// TIA Portal project "SUW_NOWE" (V18)

(* hardware
DEVICE "S7-1200 station_1"  S7-1200 Station
   slot 0: "Rack_0"  S7-1200 Rack  Rack  V1.0
   slot 1: "SUW_NOWE_CPU"  CPU 1215C DC/DC/DC  6ES7 215-1AG40-0XB0  V4.4
   slot 2: "DI 8/DQ 8x24VDC_1"  6ES7 223-1BH32-0XB0  V2.0
   slot 3: "AI 8x13BIT_1"  6ES7 231-4HF32-0XB0  V2.1
*)

// ===== PLC "SUW_NOWE_CPU"  CPU 1215C DC/DC/DC =====

VAR_GLOBAL   // PLC tag table "Default tag table"
   "System_Byte" AT %MB1 : Byte;
   "FirstScan" AT %M1.0 : Bool;
   "DiagStatusUpdate" AT %M1.1 : Bool;
   "AlwaysTRUE" AT %M1.2 : Bool;
   "AlwaysFALSE" AT %M1.3 : Bool;
   "Clock_Byte" AT %MB0 : Byte;
   "Clock_10Hz" AT %M0.0 : Bool;
   "Clock_5Hz" AT %M0.1 : Bool;
   "Clock_2.5Hz" AT %M0.2 : Bool;
   "Clock_2Hz" AT %M0.3 : Bool;
   "Clock_1.25Hz" AT %M0.4 : Bool;
   "Clock_1Hz" AT %M0.5 : Bool;
   "Clock_0.625Hz" AT %M0.6 : Bool;
   "Clock_0.5Hz" AT %M0.7 : Bool;
   "ilosc_pomp" AT %MW2 : Int;
   "moc_pomp" AT %MD4 : Real;
   "pomocnicza" AT %M8.0 : Bool;
   "bPumpsEnable" AT %M8.1 : Bool;
   "iNumPumps" AT %MW10 : Int;
   "rPumpSpeed" AT %MD12 : Real;
   "temp" AT %M8.2 : Bool;
   "temp2" AT %M8.3 : Bool;
   "bReadComplet1A" AT %M8.4 : Bool;
   "bReq1A" AT %M8.5 : Bool;
   "bReq2A" AT %M8.6 : Bool;
   "bReadComplet2A" AT %M8.7 : Bool;
   "bReq3A" AT %M9.0 : Bool;
   "bReadComplet3A" AT %M9.1 : Bool;
   "bReq2B" AT %M9.2 : Bool;
   "bReadComplet2B" AT %M9.3 : Bool;
   "bReq3" AT %M9.4 : Bool;
   "bReadComplet3" AT %M9.5 : Bool;
   "bReq5" AT %M9.6 : Bool;
   "bReadComplet5" AT %M9.7 : Bool;
END_VAR

VAR_GLOBAL   // PLC tag table "I/O"
   "bPmp1A_AutoSwitch" AT %I0.0 : Bool;   // Przełącznik AUTO pompy 1A
   "bPmp2A_AutoSwitch" AT %I0.1 : Bool;   // Przełącznik AUTO pompy 2A
   "bPmp2B_AutoSwitch" AT %I0.2 : Bool;   // Przełącznik AUTO pompy 2B
   "bPmp3_AutoSwitch" AT %I0.3 : Bool;   // Przełącznik AUTO pompy 3
   "bPmp3A_AutoSwitch" AT %I0.4 : Bool;   // Przełącznik AUTO pompy 3A
   "bPmp5_AutoSwitch" AT %I0.5 : Bool;   // Przełącznik AUTO pompy 5
   "bPmp1A_ManualSwitch" AT %I1.0 : Bool;   // Przełącznik ręczny pompy 1A
   "bPmp2A_ManualSwitch" AT %I1.1 : Bool;   // Przełącznik ręczny pompy 2A
   "bPmp2B_ManualSwitch" AT %I1.2 : Bool;   // Przełącznik ręczny pompy 2B
   "bPmp3_ManualSwitch" AT %I1.3 : Bool;   // Przełącznik ręczny pompy 3
   "bPmp3A_ManualSwitch" AT %I1.4 : Bool;   // Przełącznik ręczny pompy 3A
   "bPmp5_ManualSwitch" AT %I1.5 : Bool;   // Przełącznik ręczny pompy 5
   "bPmp1A_RunSignal" AT %Q0.0 : Bool;   // Sygnalizacja pracy pompy 1A
   "bPmp2A_RunSignal" AT %Q0.1 : Bool;   // Sygnalizacja pracy pompy 2A
   "bPmp2B_RunSignal" AT %Q0.2 : Bool;   // Sygnalizacja pracy pompy 2B
   "bPmp3_RunSignal" AT %Q0.3 : Bool;   // Sygnalizacja pracy pompy 3
   "bPmp3A_RunSignal" AT %Q0.4 : Bool;   // Sygnalizacja pracy pompy 3A
   "bPmp5_RunSignal" AT %Q0.5 : Bool;   // Sygnalizacja pracy pompy 5
   "bPmp1A_FaultSignal" AT %Q0.6 : Bool;   // Sygnalizacja awarii pompy 1A
   "bPmp2A_FaultSignal" AT %Q0.7 : Bool;   // Sygnalizacja awarii pompy 2A
   "bPmp2B_FaultSignal" AT %Q1.0 : Bool;   // Sygnalizacja awarii pompy 2B
   "bPmp3_FaultSignal" AT %Q1.1 : Bool;   // Sygnalizacja awarii pompy 3
   "bPmp3A_FaultSignal" AT %Q8.0 : Bool;   // Sygnalizacja awarii pompy 3A
   "bPmp5_FaultSignal" AT %Q8.1 : Bool;   // Sygnalizacja awarii pompy 5
END_VAR

DATA_BLOCK "KomunikacjaFalownik1A_DB"   // DB1
{ S7_Optimized_Access := 'TRUE' }
VERSION : 0.1
// stored: InstanceOfName KomunikacjaFalownik
"KomunikacjaFalownik"
BEGIN
END_DATA_BLOCK

DATA_BLOCK "ObslugaGotowosciPompy_1A_DB"   // DB2
{ S7_Optimized_Access := 'TRUE' }
VERSION : 0.1
// stored: InstanceOfName ObslugaGotowosciPompy
"ObslugaGotowosciPompy"
BEGIN
END_DATA_BLOCK

DATA_BLOCK "ObslugaGotowosciPompy_2A_DB"   // DB3
{ S7_Optimized_Access := 'TRUE' }
VERSION : 0.1
// stored: InstanceOfName ObslugaGotowosciPompy
"ObslugaGotowosciPompy"
BEGIN
END_DATA_BLOCK

DATA_BLOCK "ObslugaGotowosciPompy_2B_DB"   // DB4
{ S7_Optimized_Access := 'TRUE' }
VERSION : 0.1
// stored: InstanceOfName ObslugaGotowosciPompy
"ObslugaGotowosciPompy"
BEGIN
END_DATA_BLOCK

DATA_BLOCK "ObslugaGotowosciPompy_3_DB"   // DB5
{ S7_Optimized_Access := 'TRUE' }
VERSION : 0.1
// stored: InstanceOfName ObslugaGotowosciPompy
"ObslugaGotowosciPompy"
BEGIN
END_DATA_BLOCK

DATA_BLOCK "ObslugaGotowosciPompy_3A_DB"   // DB6
{ S7_Optimized_Access := 'TRUE' }
VERSION : 0.1
// stored: InstanceOfName ObslugaGotowosciPompy
"ObslugaGotowosciPompy"
BEGIN
END_DATA_BLOCK

DATA_BLOCK "ObslugaWyboruPomp_DB"   // DB7
{ S7_Optimized_Access := 'TRUE' }
VERSION : 0.1
// stored: InstanceOfName ObslugaWyboruPomp
"ObslugaWyboruPomp"
BEGIN
END_DATA_BLOCK

DATA_BLOCK "AutoReady"   // DB10
{ S7_Optimized_Access := 'TRUE' }
VERSION : 0.1
   VAR
      aReadyArray : Array[1..6] of Bool;
      aPumpToActive : Array[1..6] of Bool;
      iLastRotationTime : DTL;
      aTimePump : Array[1..6] of DInt;
   END_VAR
BEGIN
END_DATA_BLOCK

DATA_BLOCK "MODBUS_SERVER"   // DB11
{ S7_Optimized_Access := 'TRUE' }
VERSION : 0.1
   VAR
      tcp : TCON_IP_v4;
   END_VAR
BEGIN
   tcp.InterfaceId := 64;
   tcp.ID := 16#1;
   tcp.RemotePort := 0;
   tcp.LocalPort := 502;
   tcp.RemoteAddress.ADDR[1] := 192;
   tcp.RemoteAddress.ADDR[2] := 168;
   tcp.RemoteAddress.ADDR[3] := 99;
   tcp.RemoteAddress.ADDR[4] := 200;
   tcp.ActiveEstablished := false;
END_DATA_BLOCK

DATA_BLOCK "KomunikacjaFalownik2A_DB"   // DB13
{ S7_Optimized_Access := 'TRUE' }
VERSION : 0.1
// stored: InstanceOfName KomunikacjaFalownik
"KomunikacjaFalownik"
BEGIN
END_DATA_BLOCK

DATA_BLOCK "KomunikacjaFalownik3A_DB"   // DB14
{ S7_Optimized_Access := 'TRUE' }
VERSION : 0.1
// stored: InstanceOfName KomunikacjaFalownik
"KomunikacjaFalownik"
BEGIN
END_DATA_BLOCK

DATA_BLOCK "KomunikacjaFalownik2B_DB"   // DB17
{ S7_Optimized_Access := 'TRUE' }
VERSION : 0.1
// stored: InstanceOfName KomunikacjaFalownik
"KomunikacjaFalownik"
BEGIN
END_DATA_BLOCK

DATA_BLOCK "KomunikacjaFalownik3_DB"   // DB18
{ S7_Optimized_Access := 'TRUE' }
VERSION : 0.1
// stored: InstanceOfName KomunikacjaFalownik
"KomunikacjaFalownik"
BEGIN
END_DATA_BLOCK

DATA_BLOCK "KomunikacjaFalownik5_DB"   // DB20
{ S7_Optimized_Access := 'TRUE' }
VERSION : 0.1
// stored: InstanceOfName KomunikacjaFalownik
"KomunikacjaFalownik"
BEGIN
END_DATA_BLOCK

DATA_BLOCK "IPBlock"   // DB30
{ S7_Optimized_Access := 'TRUE' }
VERSION : 0.1
   VAR RETAIN
      IP1A : Array[1..4] of Byte;
      IP2A : Array[1..4] of Byte;
      IP2B : Array[1..4] of Byte;
      IP3 : Array[1..4] of Byte;
      IP3A : Array[1..4] of Byte;
      IP5 : Array[1..4] of Byte;
      IPBudynek : Array[1..4] of Byte;
      IPRozdzielnia : Array[1..4] of Byte;
      IPKosiby : Array[1..4] of Byte;
   END_VAR
BEGIN
   IP1A[1] := 192;
   IP1A[2] := 168;
   IP1A[3] := 99;
   IP1A[4] := 111;
   IP2A[1] := 192;
   IP2A[2] := 168;
   IP2A[3] := 99;
   IP2A[4] := 112;
END_DATA_BLOCK

DATA_BLOCK "Studnia1A"   // DB31
{ S7_Optimized_Access := 'FALSE' }
VERSION : 0.1
   VAR
      CONTROL_WORD : Int;   // Słowo sterujące dla falownika
      SETPOINT_R : Real;   // Setpoint w procentach
      SETPOINT : Int;   // Setpoint w wartości dla falownika 0-8333 dla predkości 0-3000 rpm
      STATUS_WORD : Int;   // Słowo statusowe falownika
      ACTUAL_VALUE : Int;   // Aktualna wartość z falownika
      POWER : Int;   // Moc pompy w kW [*0,01]
      MOTOR_CURRENT : Int;   // Prąd pompy w A [*0,01]
      HEATSNK_TEMP : Int;   // Temperatura radiatora w C
      INVERTER_TERM : Int;   // Status termiczny invertera
      ANALOGIN_53 : Int;   // Pętla analogowa 4-20mA (poziom)
      ALARM_WORD : Word;   // Słowo alarmowe
      ALARM_WORD_1 : Word;   // Słowo alarmowe
      ALARM_WORD_2 : Word;   // Słowo alarmowe
      WARNING_WORD : Word;   // Słowo ostrzeżenia
      WARNING_WORD_1 : Word;   // Słowo ostrzeżenia
      WARNING_WORD_2 : Word;   // Słowo ostrzeżenia
      STATUS : Word;   // Status pompy wg. rozpiski
      DONE : Bool;   // Poprawne wykonaie transmisji
      ERROR : Bool;   // Błąd wykonania transmisji
      BUSSY : Bool;   // Port zajęty
      CONNECT_ERROR : Word;   // Kod błedu
      RUN_TIME : DInt;   // Czas pracy w minutach
      RUN_COUNTER : DInt;   // Ilość załączeń
      SCADA_AUTO : Bool;   // Przełącznik pracy automatycznej 1 - zezwolenie 0 odstawienie
      SCADA_RUN : Bool;   // Sygnał załączenia ze scada
      SYSTEM_RUN : Bool;   // Sygnał załączenia przez system
      FAULT_RESET : Bool;   // Reset awarii
      WATER_LEVEL : Real;   // Poziom w studni w metrach
   END_VAR
BEGIN
END_DATA_BLOCK

DATA_BLOCK "Studnia2A"   // DB32
{ S7_Optimized_Access := 'FALSE' }
VERSION : 0.1
   VAR
      CONTROL_WORD : Int;
      SETPOINT_R : Real;
      SETPOINT : Int;
      STATUS_WORD : Int;
      ACTUAL_VALUE : Int;
      POWER : Int;
      MOTOR_CURRENT : Int;
      HEATSNK_TEMP : Int;
      INVERTER_TERM : Int;
      ANALOGIN_53 : Int;
      ALARM_WORD : Word;
      ALARM_WORD_1 : Word;
      ALARM_WORD_2 : Word;
      WARNING_WORD : Word;
      WARNING_WORD_1 : Word;
      WARNING_WORD_2 : Word;
      STATUS : Word;
      DONE : Bool;
      ERROR : Bool;
      BUSSY : Bool;
      CONNECT_ERROR : Word;
      RUN_TIME : DInt;
      RUN_COUNTER : DInt;
      SCADA_AUTO : Bool;
      SCADA_RUN : Bool;
      SYSTEM_RUN : Bool;
      FAULT_RESET : Bool;
      WATER_LEVEL : Real;   // Poziom w studni w metrach
   END_VAR
BEGIN
END_DATA_BLOCK

DATA_BLOCK "Studnia2B"   // DB33
{ S7_Optimized_Access := 'FALSE' }
VERSION : 0.1
   VAR
      CONTROL_WORD : Int;
      SETPOINT_R : Real;
      SETPOINT : Int;
      STATUS_WORD : Int;
      ACTUAL_VALUE : Int;
      POWER : Int;
      MOTOR_CURRENT : Int;
      HEATSNK_TEMP : Int;
      INVERTER_TERM : Int;
      ANALOGIN_53 : Int;
      ALARM_WORD : Word;
      ALARM_WORD_1 : Word;
      ALARM_WORD_2 : Word;
      WARNING_WORD : Word;
      WARNING_WORD_1 : Word;
      WARNING_WORD_2 : Word;
      STATUS : Word;
      DONE : Bool;
      ERROR : Bool;
      BUSSY : Bool;
      CONNECT_ERROR : Word;
      RUN_TIME : DInt;
      RUN_COUNTER : DInt;
      SCADA_AUTO : Bool;
      SCADA_RUN : Bool;
      SYSTEM_RUN : Bool;
      FAULT_RESET : Bool;
      WATER_LEVEL : Real;   // Poziom w studni w metrach
   END_VAR
BEGIN
END_DATA_BLOCK

DATA_BLOCK "Studnia3"   // DB34
{ S7_Optimized_Access := 'FALSE' }
VERSION : 0.1
   VAR
      CONTROL_WORD : Int;
      SETPOINT_R : Real;
      SETPOINT : Int;
      STATUS_WORD : Int;
      ACTUAL_VALUE : Int;
      POWER : Int;
      MOTOR_CURRENT : Int;
      HEATSNK_TEMP : Int;
      INVERTER_TERM : Int;
      ANALOGIN_53 : Int;
      ALARM_WORD : Word;
      ALARM_WORD_1 : Word;
      ALARM_WORD_2 : Word;
      WARNING_WORD : Word;
      WARNING_WORD_1 : Word;
      WARNING_WORD_2 : Word;
      STATUS : Word;
      DONE : Bool;
      ERROR : Bool;
      BUSSY : Bool;
      CONNECT_ERROR : Word;
      RUN_TIME : DInt;
      RUN_COUNTER : DInt;
      SCADA_AUTO : Bool;
      SCADA_RUN : Bool;
      SYSTEM_RUN : Bool;
      FAULT_RESET : Bool;
      WATER_LEVEL : Real;   // Poziom w studni w metrach
   END_VAR
BEGIN
END_DATA_BLOCK

DATA_BLOCK "Studnia3A"   // DB35
{ S7_Optimized_Access := 'FALSE' }
VERSION : 0.1
   VAR
      CONTROL_WORD : Int;   // Słowo sterujące dla falownika
      SETPOINT_R : Real;   // Setpoint w procentach
      SETPOINT : Int;   // Setpoint w wartości dla falownika 0-8333 dla predkości 0-3000 rpm
      STATUS_WORD : Int;   // Słowo statusowe falownika
      ACTUAL_VALUE : Int;   // Aktualna wartość z falownika
      POWER : Int;   // Moc pompy w kW [*0,01]
      MOTOR_CURRENT : Int;   // Prąd pompy w A [*0,01]
      HEATSNK_TEMP : Int;   // Temperatura radiatora w C
      INVERTER_TERM : Int;   // Status termiczny invertera
      ANALOGIN_53 : Int;   // Pętla analogowa 4-20mA (poziom)
      ALARM_WORD : Word;   // Słowo alarmowe
      ALARM_WORD_1 : Word;   // Słowo alarmowe
      ALARM_WORD_2 : Word;   // Słowo alarmowe
      WARNING_WORD : Word;   // Słowo ostrzeżenia
      WARNING_WORD_1 : Word;   // Słowo ostrzeżenia
      WARNING_WORD_2 : Word;   // Słowo ostrzeżenia
      STATUS : Word;   // Status pompy wg. rozpiski
      DONE : Bool;   // Poprawne wykonaie transmisji
      ERROR : Bool;   // Błąd wykonania transmisji
      BUSSY : Bool;   // Port zajęty
      CONNECT_ERROR : Word;   // Kod błedu
      RUN_TIME : DInt;   // Czas pracy w minutach
      RUN_COUNTER : DInt;   // Ilość załączeń
      SCADA_AUTO : Bool;   // Przełącznik pracy automatycznej 1 - zezwolenie 0 odstawienie
      SCADA_RUN : Bool;   // Sygnał załączenia ze scada
      SYSTEM_RUN : Bool;   // Sygnał załączenia przez system
      FAULT_RESET : Bool;   // Reset awarii
      WATER_LEVEL : Real;   // Poziom w studni w metrach
   END_VAR
BEGIN
END_DATA_BLOCK

DATA_BLOCK "Studnia5"   // DB36
{ S7_Optimized_Access := 'FALSE' }
VERSION : 0.1
   VAR
      CONTROL_WORD : Int;   // Słowo sterujące dla falownika
      SETPOINT_R : Real;   // Setpoint w procentach
      SETPOINT : Int;   // Setpoint w wartości dla falownika 0-8333 dla predkości 0-3000 rpm
      STATUS_WORD : Int;   // Słowo statusowe falownika
      ACTUAL_VALUE : Int;   // Aktualna wartość z falownika
      POWER : Int;   // Moc pompy w kW [*0,01]
      MOTOR_CURRENT : Int;   // Prąd pompy w A [*0,01]
      HEATSNK_TEMP : Int;   // Temperatura radiatora w C
      INVERTER_TERM : Int;   // Status termiczny invertera
      ANALOGIN_53 : Int;   // Pętla analogowa 4-20mA (poziom)
      ALARM_WORD : Word;   // Słowo alarmowe
      ALARM_WORD_1 : Word;   // Słowo alarmowe
      ALARM_WORD_2 : Word;   // Słowo alarmowe
      WARNING_WORD : Word;   // Słowo ostrzeżenia
      WARNING_WORD_1 : Word;   // Słowo ostrzeżenia
      WARNING_WORD_2 : Word;   // Słowo ostrzeżenia
      STATUS : Word;   // Status pompy wg. rozpiski
      DONE : Bool;   // Poprawne wykonaie transmisji
      ERROR : Bool;   // Błąd wykonania transmisji
      BUSSY : Bool;   // Port zajęty
      CONNECT_ERROR : Word;   // Kod błedu
      RUN_TIME : DInt;   // Czas pracy w minutach
      RUN_COUNTER : DInt;   // Ilość załączeń
      SCADA_AUTO : Bool;   // Przełącznik pracy automatycznej 1 - zezwolenie 0 odstawienie
      SCADA_RUN : Bool;   // Sygnał załączenia ze scada
      SYSTEM_RUN : Bool;   // Sygnał załączenia przez system
      FAULT_RESET : Bool;   // Reset awarii
      WATER_LEVEL : Real;   // Poziom w studni w metrach
   END_VAR
BEGIN
END_DATA_BLOCK

DATA_BLOCK "ZbiornikKosiby"   // DB40
{ S7_Optimized_Access := 'FALSE' }
VERSION : 0.1
   VAR
      iPoziomKosiby : Int;
      rPoziomKosiby : Real;
      rPoziomTest : Real;
   END_VAR
BEGIN
END_DATA_BLOCK

// folder: System blocks/Program resources

DATA_BLOCK "IEC_Timer_0_DB"   // DB9
{ S7_Optimized_Access := 'TRUE' }
AUTHOR : Simatic
FAMILY : IEC
NAME : IEC_TMR
VERSION : 1.0
// stored: InstanceOfName IEC_TIMER
"IEC_TIMER"
BEGIN
END_DATA_BLOCK

DATA_BLOCK "IEC_Timer_0_DB_1"   // DB12
{ S7_Optimized_Access := 'TRUE' }
AUTHOR : Simatic
FAMILY : IEC
NAME : IEC_TMR
VERSION : 1.0
// stored: InstanceOfName IEC_TIMER
"IEC_TIMER"
BEGIN
END_DATA_BLOCK

DATA_BLOCK "IEC_Timer_0_DB_2"   // DB15
{ S7_Optimized_Access := 'TRUE' }
AUTHOR : Simatic
FAMILY : IEC
NAME : IEC_TMR
VERSION : 1.0
// stored: InstanceOfName IEC_TIMER
"IEC_TIMER"
BEGIN
END_DATA_BLOCK

DATA_BLOCK "IEC_Timer_0_DB_3"   // DB16
{ S7_Optimized_Access := 'TRUE' }
AUTHOR : Simatic
FAMILY : IEC
NAME : IEC_TMR
VERSION : 1.0
// stored: InstanceOfName IEC_TIMER
"IEC_TIMER"
BEGIN
END_DATA_BLOCK

DATA_BLOCK "IEC_Timer_0_DB_4"   // DB19
{ S7_Optimized_Access := 'TRUE' }
AUTHOR : Simatic
FAMILY : IEC
NAME : IEC_TMR
VERSION : 1.0
// stored: InstanceOfName IEC_TIMER
"IEC_TIMER"
BEGIN
END_DATA_BLOCK

// folder: (top level)

FUNCTION_BLOCK "KomunikacjaFalownik"   // FB1, SCL
{ S7_Optimized_Access := 'TRUE' }
VERSION : 0.1
   VAR_INPUT
      bReq : Bool;   // Żądanie transmisji
      bDisconnect : Bool;   // Rozłączenie
      connID : Conn_Ouc;   // ID urządzenia
      ADDR : Array[1..4] of Byte;   // Adres IP
      wDriveControl : Word;   // Słowo sterujące falownika
      iSetpoint : Int;   // Wartość zadana falownika
      iDriverID : USInt;
   END_VAR
   VAR_OUTPUT
      bDone : Bool;
      bError : Bool;
      wStatus : Word;
      wDriveStatus : Word;
      aDriveInfo : Array[0..8] of Word;
   END_VAR
   VAR_IN_OUT
      bReadComplete : Bool;
   END_VAR
   VAR
      iStep : Int;
      mbClient : MB_CLIENT;
      connStruct : TCON_IP_v4;
   END_VAR
   VAR_TEMP
      dataPtr : Variant;
   END_VAR
   // connStruct.ActiveEstablished := true;
   // connStruct.InterfaceId := 64;
BEGIN
       // Konfiguracja połączenia
       #connStruct.RemoteAddress.ADDR := #ADDR;
       #connStruct.RemotePort := 502;
       #connStruct.ID := #connID;

       // Sekwencyjne wykonywanie zapytań
       CASE #iStep OF
               // 0: Start transmisji
           0:
               IF #bReq THEN
                   #iStep := 1;
                   #bReadComplete := FALSE;
               END_IF;

               // 1: Zapis słowa sterującego do falownika
           1:

               #mbClient.MB_Unit_ID := #iDriverID;
               #mbClient(
                         REQ := TRUE,
                         DISCONNECT := #bDisconnect,
                         MB_MODE := 106, // Write Multiple Registers
                         MB_DATA_ADDR := 101,
                         MB_DATA_LEN :=1,
                         MB_DATA_PTR := #wDriveControl, // Wskaźnik do zmiennych sterujących
                         CONNECT := #connStruct,
                         DONE => #bDone,
                         ERROR => #bError,
                         STATUS => #wStatus



               );
               IF #bDone THEN
                   #iStep := 2;
               ELSIF #bError THEN
                   #iStep := 99; // Przeskok do błędu
               END_IF;

               // 1: Zapis setpointu do falownika
               // 
           2:
               #mbClient.MB_Unit_ID := #iDriverID;
               #mbClient(
                         REQ := TRUE,
                         DISCONNECT := #bDisconnect,
                         MB_MODE := 106, // Write Multiple Registers
                         MB_DATA_ADDR := 104,
                         MB_DATA_LEN := 1,
                         MB_DATA_PTR := #iSetpoint, // Wskaźnik do zmiennych sterujących
                         CONNECT := #connStruct,
                         DONE => #bDone,
                         ERROR => #bError,
                         STATUS => #wStatus



               );
               IF #bDone THEN
                   #iStep := 3;
               ELSIF #bError THEN
                   #iStep := 99; // Przeskok do błędu
               END_IF;

               // 3: Odczyt statusu falownika
           3:
               #mbClient.MB_Unit_ID := #iDriverID;
               #mbClient(
                         REQ := TRUE,
                         DISCONNECT := #bDisconnect,
                         MB_MODE := 103, // Read Holding Registers
                         MB_DATA_ADDR := 201,
                         MB_DATA_LEN := 1,
                         MB_DATA_PTR := #wDriveStatus,
                         CONNECT := #connStruct,
                         DONE => #bDone,
                         ERROR => #bError,
                         STATUS => #wStatus
               );
               IF #bDone THEN
                   #iStep := 4;
               ELSIF #bError THEN
                   #iStep := 99;
               END_IF;

               // 4: Odczyt dodatkowych danych falownika
           4:
               #mbClient.MB_Unit_ID := #iDriverID;
               #mbClient(
                         REQ := TRUE,
                         DISCONNECT := #bDisconnect,
                         MB_MODE := 103,
                         MB_DATA_ADDR := 2911,
                         MB_DATA_LEN := 9,
                         MB_DATA_PTR := #aDriveInfo,
                         CONNECT := #connStruct,
                         DONE => #bDone,
                         ERROR => #bError,
                         STATUS => #wStatus
               );
               IF #bDone THEN
                   #iStep := 10;
               ELSIF #bError THEN
                   #iStep := 99;
               END_IF;



               // 10: Zakończenie odczytu
           10:
               #bReadComplete := TRUE;
               #iStep := 0; // Reset do początku

               // 99: Obsługa błędu
           99:
               #bReadComplete := TRUE;
               #bError := TRUE;
               #iStep := 0; // Reset do początku
       END_CASE;
END_FUNCTION_BLOCK

FUNCTION_BLOCK "ObslugaWyboruPomp"   // FB2, SCL
{ S7_Optimized_Access := 'TRUE' }
VERSION : 0.1
   VAR_INPUT
      iRequestedPumps : Int;   // Liczba pomp do uruchomienia
      aPumpReady : Array[1..6] of Bool;   // Gotowość pomp
      dPumpRuntime : Array[1..6] of DInt;   // Czas pracy pomp w minutach
      iCurrentTime : DTL;   // Aktualny czas systemowy
      iRotationTime : Time := T#4h;
   END_VAR
   VAR_IN_OUT
      iActivePumps : Array[1..6] of Bool;   // Aktywne pompy
      bNotEnoughPumpsAvailable : Bool;   // Flaga braku wymaganej liczby pomp
      iLastRotationTime : DTL;
   END_VAR
   VAR
      bRotationRequired : Bool;
      iPumpPriority : Array[1..6] of Int;   // Posortowane indeksy pomp wg czasu pracy
      minRuntime : DInt;
      minPumpIdx : Int;
      i : Int;
      j : Int;
      minIdx : Int;
      activeCount : Int;
      availableCount : Int;
      eligiblePumps : Array[1..6] of Bool;
      tempRuntime : Int;
      tempIdx : Int;
      selectedPump : Int;   // Posortowane indeksy pomp wg czasu pracy
      conflict : Bool;
      n : Int;
   END_VAR
BEGIN
   // Resetowanie tablicy aktywnych pomp
   FOR #i := 1 TO 6 DO
       #iActivePumps[#i] := FALSE;
   END_FOR;

   #bNotEnoughPumpsAvailable := FALSE; // Reset flagi

   // Sprawdzenie, czy należy przeprowadzić rotację pomp
   IF (#iRequestedPumps > 0) AND ((#iCurrentTime - #iLastRotationTime) >= #iRotationTime) THEN
       #iLastRotationTime := #iCurrentTime; // Aktualizacja czasu rotacji
       #bRotationRequired := TRUE;
   END_IF;

   // Filtrowanie dostępnych pomp
   #availableCount := 0;
   FOR #i := 1 TO 6 DO
       #eligiblePumps[#i] := #aPumpReady[#i];  // Czy pompa jest gotowa
       //#iPumpPriority[#i] := #i;  // Przechowujemy numer pompy

       IF #eligiblePumps[#i] THEN
           #availableCount := #availableCount + 1;
       END_IF;
   END_FOR;

   // Sortowanie pomp po czasie pracy, od najmniejszego do największego
   IF #bRotationRequired THEN
       FOR #i := 1 TO 5 DO
           #minIdx := #i;

           FOR #j := #i + 1 TO 6 DO
               IF #dPumpRuntime[#iPumpPriority[#j]] < #dPumpRuntime[#iPumpPriority[#minIdx]] THEN
                   #minIdx := #j;
               END_IF;
           END_FOR;

           // Zamiana miejscami
           IF #minIdx <> #i THEN
               #tempIdx := #iPumpPriority[#i];
               #iPumpPriority[#i] := #iPumpPriority[#minIdx];
               #iPumpPriority[#minIdx] := #tempIdx;
           END_IF;
       END_FOR;
       #bRotationRequired := FALSE;
   END_IF;

   // Wybór pomp, unikając konfliktów (2A/2B i 3/3A)
   #activeCount := 0;
   FOR #i := 1 TO 6 DO
       #selectedPump := #iPumpPriority[#i];

       IF (#activeCount < #iRequestedPumps) AND #eligiblePumps[#selectedPump] THEN
           // Sprawdzenie konfliktów 2A/2B i 3/3A
           #conflict := FALSE;

           IF ((#selectedPump = 2) AND (#iActivePumps[3])) OR
               ((#selectedPump = 3) AND (#iActivePumps[2])) OR
               ((#selectedPump = 4) AND (#iActivePumps[5])) OR
               ((#selectedPump = 5) AND (#iActivePumps[4])) THEN
               #conflict := TRUE;
           END_IF;

           // Jeśli nie ma konfliktu, aktywujemy pompę
           IF NOT #conflict THEN
               #iActivePumps[#selectedPump] := TRUE;
               #activeCount := #activeCount + 1;
               #eligiblePumps[#selectedPump] := FALSE; // Wykluczenie pompy z kolejnej pętli
           END_IF;
       END_IF;
   END_FOR;

   // Sprawdzenie, czy dostępnych pomp było za mało
   #bNotEnoughPumpsAvailable := (#activeCount < #iRequestedPumps);
END_FUNCTION_BLOCK

FUNCTION_BLOCK "ObslugaGotowosciPompy"   // FB3, SCL
{ S7_Optimized_Access := 'TRUE' }
VERSION : 0.1
   VAR_INPUT
      bAutoMode : Bool;   // Tryb automatyczny
      bManualMode : Bool;   // Tryb ręczny
      bStartCmd : Bool;   // Start pompy (tylko w automacie)
      iDriveStatus : Int;   // Reset awarii
      rSpeedSetpoint : Real;   // Status falownika (odczytany)
      rWellLevel : Real;   // Poziom wody w studni
      rDryRunLevel : Real;   // Poziom sucho biegu
      rDryRunHyst : Real;   // Histereza sucho biegu
      bComFault : Bool;   // Błąd komunikacji
   END_VAR
   VAR_OUTPUT
      iControlWord : Int;   // Słowo sterujące dla falownika
      iSetpoint : Int;   // Punkt pracy pompy (0-8333)
      iPumpStatus : Int;   // Status pompy
      bPumpReady : Bool;   // Gotowość do pracy auto
      bPumpFaultLED : Bool;   // Sygnalizacja awari
      bPumpRuningLED : Bool;   // Sygnalizacja pracy
   END_VAR
   VAR_IN_OUT
      iStartCounter : DInt;   // Licznik załączeń
      bFaultReset : Bool;   // Zadana prędkość pompy (77-90%)
      iRunTime : DInt;   // Licznik czasu pracy (minuty)
   END_VAR
   VAR
      tResetTimer : TON_TIME;   // Timer do kasowania resetu
      bPrevRunning : Bool;   // Poprzedni stan pracy (dla licznika startów)
      iMinutesCounter : DInt;   // Pomocniczy licznik minut
      tRunTimeTimer : TON_TIME;
   END_VAR
   VAR_TEMP
      bPumpRunning : Bool;   // Czy pompa pracuje
      bPumpFault : Bool;   // Awaria pompy
      bWarning : Bool;   // Ostrzeżenie
      bDryRun : Bool;   // Sucho bieg
      bPumpComFault : Bool;   // Błąd komunikacji
   END_VAR
BEGIN
   // =======================
   // 1. Odczyt statusu falownika
   // =======================
   // 
   #bPumpRunning := (#iDriveStatus AND 16#40) > 0;  // Bit 6 - Praca
   #bPumpFault := (#iDriveStatus AND 16#400) > 0;   // Bit 10 - Awaria
   #bWarning := (#iDriveStatus AND 16#800) > 0;     // Bit 11 - Ostrzeżenie
   #bPumpComFault := #bComFault;
   //
   // =======================
   // 2. Obsługa sucho biegu
   // =======================
   // 
   IF #rWellLevel < #rDryRunLevel THEN
       #bDryRun := TRUE;
   ELSIF #rWellLevel > (#rDryRunLevel + #rDryRunHyst) THEN
       #bDryRun := FALSE;
   END_IF;

   // =======================
   // 3. Określenie warunku startu
   // =======================
   IF (#bAutoMode AND #bStartCmd) OR #bManualMode THEN
       IF NOT #bPumpFault AND NOT #bDryRun AND NOT #bComFault THEN
           #iControlWord := 16#3; // Bit 0 = 1, Bit 1 (Start) = 1
       ELSE
           #iControlWord := 16#1; // Bit 0 = 1, Bit 1 (Start) = 0
       END_IF;
   ELSE
       #iControlWord := 16#1; // Postój
   END_IF;

   // =======================
   // 4. Obsługa resetu awarii
   // =======================
   IF #bFaultReset THEN
       #iControlWord := #iControlWord OR 16#4; // Ustawienie resetu awarii (Bit 2 = 1)
       #tResetTimer(IN := TRUE,
                    PT := T#3S);
   ELSE
       #tResetTimer(IN := FALSE,PT := T#3S);
   END_IF;

   // Po 3 sekundach kasujemy bit resetu
   IF #tResetTimer.Q THEN
       #iControlWord := #iControlWord AND NOT 16#4; // Kasowanie bitu resetu (Bit 2 = 0)
   END_IF;

   // =======================
   // 5. Przeliczenie setpointa (prędkości pompy)
   // =======================
   #iSetpoint := REAL_TO_INT((#rSpeedSetpoint / 100.0) * 8333.0);

   // =======================
   // 6. Liczniki czasu pracy i załączeń
   // =======================

   IF #bPumpRunning THEN
       #tRunTimeTimer(IN := TRUE,
                     PT := T#60S); // Start timera 60s
   ELSE
       #tRunTimeTimer(IN := FALSE, PT := T#60S);
   END_IF;

   IF #tRunTimeTimer.Q THEN
       #iRunTime := #iRunTime + 1; // Po każdej minucie zwiększamy licznik
       #tRunTimeTimer(IN := FALSE, PT := T#60S); // Resetujemy timer
   END_IF;

   // Licznik załączeń
   IF NOT #bPrevRunning AND #bPumpRunning THEN
       #iStartCounter := #iStartCounter + 1;
   END_IF;
   #bPrevRunning := #bPumpRunning;

   // =======================
   // 7. Tworzenie statusu pompy
   // =======================
   #iPumpStatus := 0;

   // Postój auto / ręka
   IF NOT #bPumpRunning THEN
       IF #bAutoMode THEN
           #iPumpStatus := #iPumpStatus OR 16#1; // Bit 0 - Postój auto
       ELSE
           #iPumpStatus := #iPumpStatus OR 16#2; // Bit 1 - Postój ręka
       END_IF;
   END_IF;

   // Praca auto / ręka
   IF #bPumpRunning THEN
       IF #bAutoMode THEN
           #iPumpStatus := #iPumpStatus OR 16#4; // Bit 2 - Praca auto
       ELSE
           #iPumpStatus := #iPumpStatus OR 16#8; // Bit 3 - Praca ręka
       END_IF;
   END_IF;

   // Sucho bieg
   IF #bDryRun THEN
       #iPumpStatus := #iPumpStatus OR 16#10; // Bit 4 - Sucho bieg
   END_IF;

   // Awaria
   IF #bPumpFault THEN
       #iPumpStatus := #iPumpStatus OR 16#20; // Bit 5 - Awaria Falownik
   END_IF;

   // Ostrzeżenie
   IF #bWarning THEN
       #iPumpStatus := #iPumpStatus OR 16#40; // Bit 6 - Ostrzeżenie
   END_IF;

   // Brak komunikacji
   IF #bPumpComFault THEN
       #iPumpStatus := #iPumpStatus OR 16#80; // Bit 7 - Brak Komunikacji
   END_IF;
   // =======================
   // 8. Tworzenie informacji o gotowości pompy do pracy auto, awari i pracy
   // =======================
   #bPumpReady := #bAutoMode AND NOT #bPumpFault AND NOT #bPumpComFault AND NOT #bDryRun;
   #bPumpFaultLED := #bPumpFault OR #bPumpComFault OR #bDryRun;
   #bPumpRuningLED := #bPumpRunning;
END_FUNCTION_BLOCK

FUNCTION "ObslugaZbiornika" : Void   // FC1, SCL
{ S7_Optimized_Access := 'TRUE' }
VERSION : 0.1
   VAR_INPUT
      rTankLevel : Real;   // Aktualny poziom zbiornika
      rLevelMin : Real;   // Poziom minimalny
      rLevelMax : Real;   // Poziom maksymalny
      rHysteresis : Real;   // Histereza załączenia
   END_VAR
   VAR_IN_OUT
      iLastPumpCount : Int;
   END_VAR
   VAR_TEMP
      aUpperLimits : Array[1..4] of Real;   // Zapamiętana liczba pomp z poprzedniego cyklu
   END_VAR
BEGIN
       // Obliczenie górnych granic zakresów dla 4→0 pomp
       #aUpperLimits[1] := #rLevelMin + (#rLevelMax - #rLevelMin) * 0.25; // dla 4 pomp
       #aUpperLimits[2] := #rLevelMin + (#rLevelMax - #rLevelMin) * 0.50; // dla 3 pomp
       #aUpperLimits[3] := #rLevelMin + (#rLevelMax - #rLevelMin) * 0.75; // dla 2 pomp
       #aUpperLimits[4] := #rLevelMax;                                  // dla 1 pompy

       CASE #iLastPumpCount OF
           0:
               // załączenie 1 pompy dopiero po spadku < próg 1 - histereza
               IF #rTankLevel < (#aUpperLimits[4] - #rHysteresis) THEN
                   #iLastPumpCount := 1;
               END_IF;

           1:
               IF #rTankLevel >= #aUpperLimits[4] THEN
                   #iLastPumpCount := 0;
               ELSIF #rTankLevel < (#aUpperLimits[3] - #rHysteresis) THEN
                   #iLastPumpCount := 2;
               END_IF;

           2:
               IF #rTankLevel >= #aUpperLimits[3] THEN
                   #iLastPumpCount := 1;
               ELSIF #rTankLevel < (#aUpperLimits[2] - #rHysteresis) THEN
                   #iLastPumpCount := 3;
               END_IF;

           3:
               IF #rTankLevel >= #aUpperLimits[2] THEN
                   #iLastPumpCount := 2;
               ELSIF #rTankLevel < (#aUpperLimits[1] - #rHysteresis) THEN
                   #iLastPumpCount := 4;
               END_IF;

           4:
               IF #rTankLevel >= #aUpperLimits[1] THEN
                   #iLastPumpCount := 3;
               END_IF;
       END_CASE;
END_FUNCTION

FUNCTION "ObslugaPomp" : Void   // FC2, LAD
{ S7_Optimized_Access := 'TRUE' }
VERSION : 0.1
   VAR_TEMP
      SYS_DTL : DTL;
      ret : Int;
   END_VAR
   VAR CONSTANT
      iLastTimeRotation : DTL;
   END_VAR
BEGIN

REGION Network 1
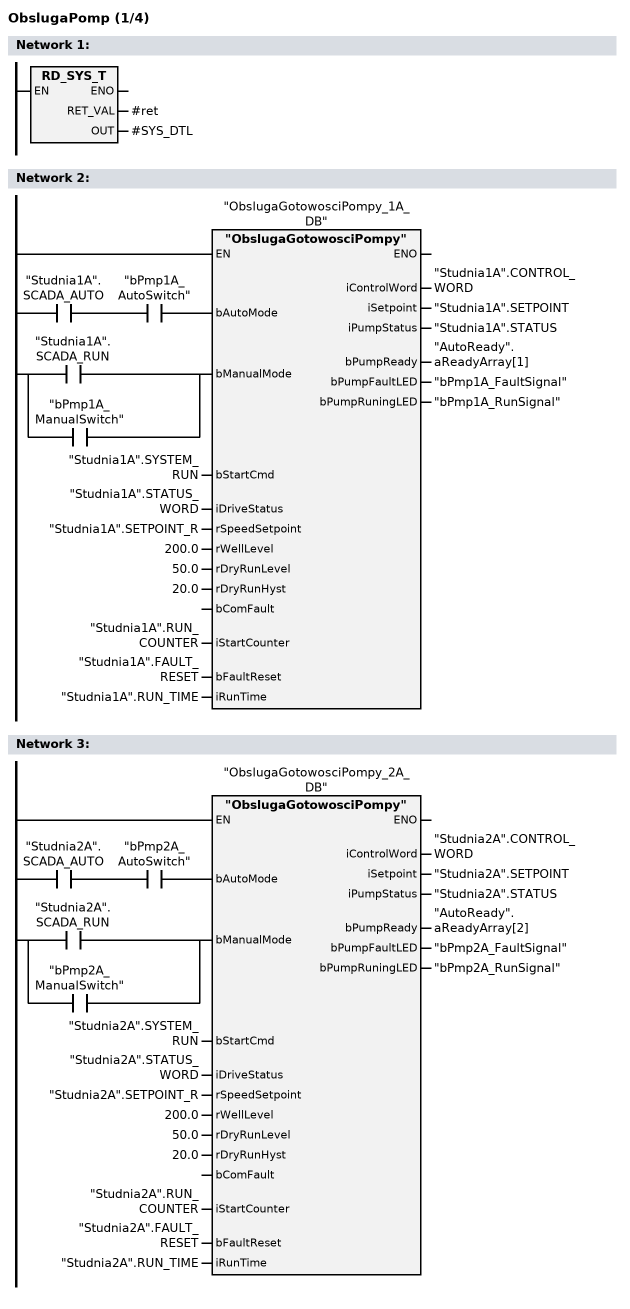
   #ret := RD_SYS_T(OUT => #SYS_DTL);
END_REGION

REGION Network 2
   RUNG wire#powerrail
      "ObslugaGotowosciPompy_1A_DB"(bAutoMode := wire#w1, bManualMode := wire#w2, bStartCmd := "Studnia1A".SYSTEM_RUN, iDriveStatus := "Studnia1A".STATUS_WORD, rSpeedSetpoint := "Studnia1A".SETPOINT_R, rWellLevel := 200.0, rDryRunLevel := 50.0, rDryRunHyst := 20.0, bComFault :=, iStartCounter := "Studnia1A".RUN_COUNTER, bFaultReset := "Studnia1A".FAULT_RESET, iRunTime := "Studnia1A".RUN_TIME, iControlWord => "Studnia1A".CONTROL_WORD, iSetpoint => "Studnia1A".SETPOINT, iPumpStatus => "Studnia1A".STATUS, bPumpReady => "AutoReady".aReadyArray[1], bPumpFaultLED => "bPmp1A_FaultSignal", bPumpRuningLED => "bPmp1A_RunSignal")
   END_RUNG
   RUNG wire#powerrail
      Contact( "Studnia1A".SCADA_AUTO )
      Contact( "bPmp1A_AutoSwitch" )
   END_RUNG wire#w1
   RUNG wire#powerrail
      Contact( "Studnia1A".SCADA_RUN )
   END_RUNG wire#w2
   RUNG wire#powerrail
      Contact( "bPmp1A_ManualSwitch" )
   END_RUNG wire#w2
   // the same network as SCL:
   "ObslugaGotowosciPompy_1A_DB"(bAutoMode := "Studnia1A".SCADA_AUTO AND "bPmp1A_AutoSwitch",   // "ObslugaGotowosciPompy"
                           bManualMode := "Studnia1A".SCADA_RUN OR "bPmp1A_ManualSwitch",
                           bStartCmd := "Studnia1A".SYSTEM_RUN,
                           iDriveStatus := "Studnia1A".STATUS_WORD,
                           rSpeedSetpoint := "Studnia1A".SETPOINT_R,
                           rWellLevel := 200.0,
                           rDryRunLevel := 50.0,
                           rDryRunHyst := 20.0,
                           iStartCounter := "Studnia1A".RUN_COUNTER,
                           bFaultReset := "Studnia1A".FAULT_RESET,
                           iRunTime := "Studnia1A".RUN_TIME,
                           iControlWord => "Studnia1A".CONTROL_WORD,
                           iSetpoint => "Studnia1A".SETPOINT,
                           iPumpStatus => "Studnia1A".STATUS,
                           bPumpReady => "AutoReady".aReadyArray[1],
                           bPumpFaultLED => "bPmp1A_FaultSignal",
                           bPumpRuningLED => "bPmp1A_RunSignal");
END_REGION

REGION Network 3
   RUNG wire#powerrail
      "ObslugaGotowosciPompy_2A_DB"(bAutoMode := wire#w1, bManualMode := wire#w2, bStartCmd := "Studnia2A".SYSTEM_RUN, iDriveStatus := "Studnia2A".STATUS_WORD, rSpeedSetpoint := "Studnia2A".SETPOINT_R, rWellLevel := 200.0, rDryRunLevel := 50.0, rDryRunHyst := 20.0, bComFault :=, iStartCounter := "Studnia2A".RUN_COUNTER, bFaultReset := "Studnia2A".FAULT_RESET, iRunTime := "Studnia2A".RUN_TIME, iControlWord => "Studnia2A".CONTROL_WORD, iSetpoint => "Studnia2A".SETPOINT, iPumpStatus => "Studnia2A".STATUS, bPumpReady => "AutoReady".aReadyArray[2], bPumpFaultLED => "bPmp2A_FaultSignal", bPumpRuningLED => "bPmp2A_RunSignal")
   END_RUNG
   RUNG wire#powerrail
      Contact( "Studnia2A".SCADA_AUTO )
      Contact( "bPmp2A_AutoSwitch" )
   END_RUNG wire#w1
   RUNG wire#powerrail
      Contact( "Studnia2A".SCADA_RUN )
   END_RUNG wire#w2
   RUNG wire#powerrail
      Contact( "bPmp2A_ManualSwitch" )
   END_RUNG wire#w2
   // the same network as SCL:
   "ObslugaGotowosciPompy_2A_DB"(bAutoMode := "Studnia2A".SCADA_AUTO AND "bPmp2A_AutoSwitch",   // "ObslugaGotowosciPompy"
                           bManualMode := "Studnia2A".SCADA_RUN OR "bPmp2A_ManualSwitch",
                           bStartCmd := "Studnia2A".SYSTEM_RUN,
                           iDriveStatus := "Studnia2A".STATUS_WORD,
                           rSpeedSetpoint := "Studnia2A".SETPOINT_R,
                           rWellLevel := 200.0,
                           rDryRunLevel := 50.0,
                           rDryRunHyst := 20.0,
                           iStartCounter := "Studnia2A".RUN_COUNTER,
                           bFaultReset := "Studnia2A".FAULT_RESET,
                           iRunTime := "Studnia2A".RUN_TIME,
                           iControlWord => "Studnia2A".CONTROL_WORD,
                           iSetpoint => "Studnia2A".SETPOINT,
                           iPumpStatus => "Studnia2A".STATUS,
                           bPumpReady => "AutoReady".aReadyArray[2],
                           bPumpFaultLED => "bPmp2A_FaultSignal",
                           bPumpRuningLED => "bPmp2A_RunSignal");
END_REGION

REGION Network 4
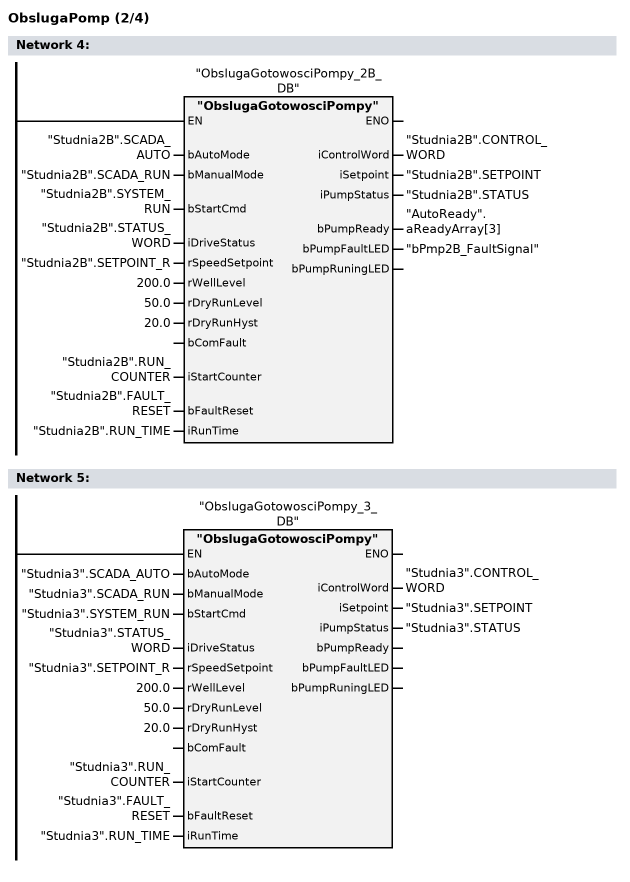
   RUNG wire#powerrail
      "ObslugaGotowosciPompy_2B_DB"(bAutoMode := "Studnia2B".SCADA_AUTO, bManualMode := "Studnia2B".SCADA_RUN, bStartCmd := "Studnia2B".SYSTEM_RUN, iDriveStatus := "Studnia2B".STATUS_WORD, rSpeedSetpoint := "Studnia2B".SETPOINT_R, rWellLevel := 200.0, rDryRunLevel := 50.0, rDryRunHyst := 20.0, bComFault :=, iStartCounter := "Studnia2B".RUN_COUNTER, bFaultReset := "Studnia2B".FAULT_RESET, iRunTime := "Studnia2B".RUN_TIME, iControlWord => "Studnia2B".CONTROL_WORD, iSetpoint => "Studnia2B".SETPOINT, iPumpStatus => "Studnia2B".STATUS, bPumpReady => "AutoReady".aReadyArray[3], bPumpFaultLED => "bPmp2B_FaultSignal", bPumpRuningLED =>)
   END_RUNG
   // the same network as SCL:
   "ObslugaGotowosciPompy_2B_DB"(bAutoMode := "Studnia2B".SCADA_AUTO,   // "ObslugaGotowosciPompy"
                           bManualMode := "Studnia2B".SCADA_RUN,
                           bStartCmd := "Studnia2B".SYSTEM_RUN,
                           iDriveStatus := "Studnia2B".STATUS_WORD,
                           rSpeedSetpoint := "Studnia2B".SETPOINT_R,
                           rWellLevel := 200.0,
                           rDryRunLevel := 50.0,
                           rDryRunHyst := 20.0,
                           iStartCounter := "Studnia2B".RUN_COUNTER,
                           bFaultReset := "Studnia2B".FAULT_RESET,
                           iRunTime := "Studnia2B".RUN_TIME,
                           iControlWord => "Studnia2B".CONTROL_WORD,
                           iSetpoint => "Studnia2B".SETPOINT,
                           iPumpStatus => "Studnia2B".STATUS,
                           bPumpReady => "AutoReady".aReadyArray[3],
                           bPumpFaultLED => "bPmp2B_FaultSignal");
END_REGION

REGION Network 5
   RUNG wire#powerrail
      "ObslugaGotowosciPompy_3_DB"(bAutoMode := "Studnia3".SCADA_AUTO, bManualMode := "Studnia3".SCADA_RUN, bStartCmd := "Studnia3".SYSTEM_RUN, iDriveStatus := "Studnia3".STATUS_WORD, rSpeedSetpoint := "Studnia3".SETPOINT_R, rWellLevel := 200.0, rDryRunLevel := 50.0, rDryRunHyst := 20.0, bComFault :=, iStartCounter := "Studnia3".RUN_COUNTER, bFaultReset := "Studnia3".FAULT_RESET, iRunTime := "Studnia3".RUN_TIME, iControlWord => "Studnia3".CONTROL_WORD, iSetpoint => "Studnia3".SETPOINT, iPumpStatus => "Studnia3".STATUS, bPumpReady =>, bPumpFaultLED =>, bPumpRuningLED =>)
   END_RUNG
   // the same network as SCL:
   "ObslugaGotowosciPompy_3_DB"(bAutoMode := "Studnia3".SCADA_AUTO,   // "ObslugaGotowosciPompy"
                           bManualMode := "Studnia3".SCADA_RUN,
                           bStartCmd := "Studnia3".SYSTEM_RUN,
                           iDriveStatus := "Studnia3".STATUS_WORD,
                           rSpeedSetpoint := "Studnia3".SETPOINT_R,
                           rWellLevel := 200.0,
                           rDryRunLevel := 50.0,
                           rDryRunHyst := 20.0,
                           iStartCounter := "Studnia3".RUN_COUNTER,
                           bFaultReset := "Studnia3".FAULT_RESET,
                           iRunTime := "Studnia3".RUN_TIME,
                           iControlWord => "Studnia3".CONTROL_WORD,
                           iSetpoint => "Studnia3".SETPOINT,
                           iPumpStatus => "Studnia3".STATUS);
END_REGION

REGION Network 6
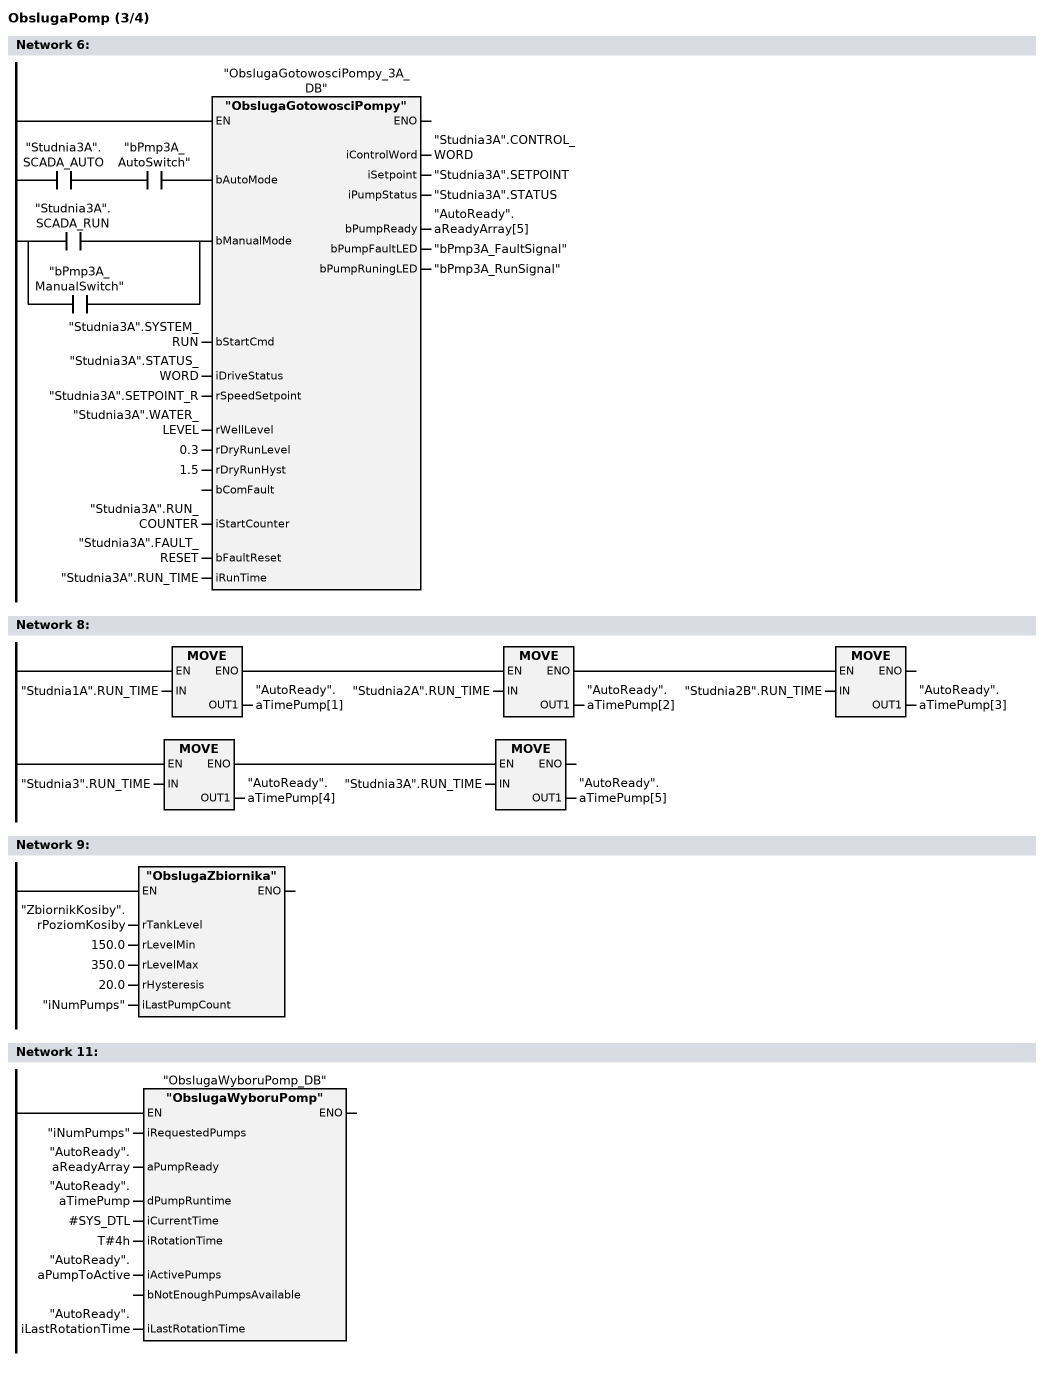
   RUNG wire#powerrail
      "ObslugaGotowosciPompy_3A_DB"(bAutoMode := wire#w1, bManualMode := wire#w2, bStartCmd := "Studnia3A".SYSTEM_RUN, iDriveStatus := "Studnia3A".STATUS_WORD, rSpeedSetpoint := "Studnia3A".SETPOINT_R, rWellLevel := "Studnia3A".WATER_LEVEL, rDryRunLevel := 0.3, rDryRunHyst := 1.5, bComFault :=, iStartCounter := "Studnia3A".RUN_COUNTER, bFaultReset := "Studnia3A".FAULT_RESET, iRunTime := "Studnia3A".RUN_TIME, iControlWord => "Studnia3A".CONTROL_WORD, iSetpoint => "Studnia3A".SETPOINT, iPumpStatus => "Studnia3A".STATUS, bPumpReady => "AutoReady".aReadyArray[5], bPumpFaultLED => "bPmp3A_FaultSignal", bPumpRuningLED => "bPmp3A_RunSignal")
   END_RUNG
   RUNG wire#powerrail
      Contact( "Studnia3A".SCADA_AUTO )
      Contact( "bPmp3A_AutoSwitch" )
   END_RUNG wire#w1
   RUNG wire#powerrail
      Contact( "Studnia3A".SCADA_RUN )
   END_RUNG wire#w2
   RUNG wire#powerrail
      Contact( "bPmp3A_ManualSwitch" )
   END_RUNG wire#w2
   // the same network as SCL:
   "ObslugaGotowosciPompy_3A_DB"(bAutoMode := "Studnia3A".SCADA_AUTO AND "bPmp3A_AutoSwitch",   // "ObslugaGotowosciPompy"
                           bManualMode := "Studnia3A".SCADA_RUN OR "bPmp3A_ManualSwitch",
                           bStartCmd := "Studnia3A".SYSTEM_RUN,
                           iDriveStatus := "Studnia3A".STATUS_WORD,
                           rSpeedSetpoint := "Studnia3A".SETPOINT_R,
                           rWellLevel := "Studnia3A".WATER_LEVEL,
                           rDryRunLevel := 0.3,
                           rDryRunHyst := 1.5,
                           iStartCounter := "Studnia3A".RUN_COUNTER,
                           bFaultReset := "Studnia3A".FAULT_RESET,
                           iRunTime := "Studnia3A".RUN_TIME,
                           iControlWord => "Studnia3A".CONTROL_WORD,
                           iSetpoint => "Studnia3A".SETPOINT,
                           iPumpStatus => "Studnia3A".STATUS,
                           bPumpReady => "AutoReady".aReadyArray[5],
                           bPumpFaultLED => "bPmp3A_FaultSignal",
                           bPumpRuningLED => "bPmp3A_RunSignal");
END_REGION

REGION Network 8
   RUNG wire#powerrail
      Move(in := "Studnia1A".RUN_TIME, out1 => "AutoReady".aTimePump[1])
      Move(in := "Studnia2A".RUN_TIME, out1 => "AutoReady".aTimePump[2])
      Move(in := "Studnia2B".RUN_TIME, out1 => "AutoReady".aTimePump[3])
   END_RUNG
   RUNG wire#powerrail
      Move(in := "Studnia3".RUN_TIME, out1 => "AutoReady".aTimePump[4])
      Move(in := "Studnia3A".RUN_TIME, out1 => "AutoReady".aTimePump[5])
   END_RUNG
   // the same network as SCL:
   "AutoReady".aTimePump[1] := "Studnia1A".RUN_TIME;
   "AutoReady".aTimePump[2] := "Studnia2A".RUN_TIME;
   "AutoReady".aTimePump[3] := "Studnia2B".RUN_TIME;
   "AutoReady".aTimePump[4] := "Studnia3".RUN_TIME;
   "AutoReady".aTimePump[5] := "Studnia3A".RUN_TIME;
END_REGION

REGION Network 9
   RUNG wire#powerrail
      "ObslugaZbiornika"(rTankLevel := "ZbiornikKosiby".rPoziomKosiby, rLevelMin := 150.0, rLevelMax := 350.0, rHysteresis := 20.0, iLastPumpCount := "iNumPumps")
   END_RUNG
   // the same network as SCL:
   "ObslugaZbiornika"(rTankLevel := "ZbiornikKosiby".rPoziomKosiby,
                      rLevelMin := 150.0,
                      rLevelMax := 350.0,
                      rHysteresis := 20.0,
                      iLastPumpCount := "iNumPumps");
END_REGION

REGION Network 11
   RUNG wire#powerrail
      "ObslugaWyboruPomp_DB"(iRequestedPumps := "iNumPumps", aPumpReady := "AutoReady".aReadyArray, dPumpRuntime := "AutoReady".aTimePump, iCurrentTime := #SYS_DTL, iRotationTime := T#4h, iActivePumps := "AutoReady".aPumpToActive, bNotEnoughPumpsAvailable :=, iLastRotationTime := "AutoReady".iLastRotationTime)
   END_RUNG
   // the same network as SCL:
   "ObslugaWyboruPomp_DB"(iRequestedPumps := "iNumPumps",   // "ObslugaWyboruPomp"
                          aPumpReady := "AutoReady".aReadyArray,
                          dPumpRuntime := "AutoReady".aTimePump,
                          iCurrentTime := #SYS_DTL,
                          iRotationTime := T#4h,
                          iActivePumps := "AutoReady".aPumpToActive,
                          iLastRotationTime := "AutoReady".iLastRotationTime);
END_REGION

REGION Network 12
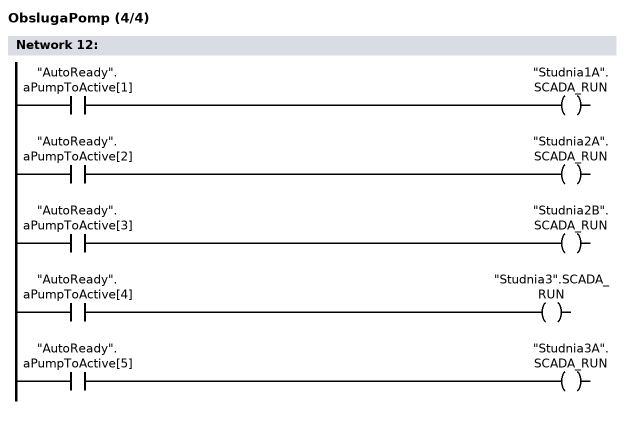
   RUNG wire#powerrail
      Contact( "AutoReady".aPumpToActive[1] )
      Coil( "Studnia1A".SCADA_RUN )
   END_RUNG
   RUNG wire#powerrail
      Contact( "AutoReady".aPumpToActive[2] )
      Coil( "Studnia2A".SCADA_RUN )
   END_RUNG
   RUNG wire#powerrail
      Contact( "AutoReady".aPumpToActive[3] )
      Coil( "Studnia2B".SCADA_RUN )
   END_RUNG
   RUNG wire#powerrail
      Contact( "AutoReady".aPumpToActive[4] )
      Coil( "Studnia3".SCADA_RUN )
   END_RUNG
   RUNG wire#powerrail
      Contact( "AutoReady".aPumpToActive[5] )
      Coil( "Studnia3A".SCADA_RUN )
   END_RUNG
   // the same network as SCL:
   "Studnia1A".SCADA_RUN := "AutoReady".aPumpToActive[1];
   "Studnia2A".SCADA_RUN := "AutoReady".aPumpToActive[2];
   "Studnia2B".SCADA_RUN := "AutoReady".aPumpToActive[3];
   "Studnia3".SCADA_RUN := "AutoReady".aPumpToActive[4];
   "Studnia3A".SCADA_RUN := "AutoReady".aPumpToActive[5];
END_REGION
END_FUNCTION

FUNCTION "ObslugaAnalogow" : Void   // FC3, SCL
{ S7_Optimized_Access := 'TRUE' }
VERSION : 0.1
BEGIN
   "Studnia3A".WATER_LEVEL := SCALE_X(MIN := 0, VALUE := NORM_X(MIN := 4000, VALUE := "Studnia3A".ANALOGIN_53, MAX := 20000), MAX := 10);
END_FUNCTION

ORGANIZATION_BLOCK "Main"   // OB1, LAD, ProgramCycle
TITLE = "Main Program Sweep (Cycle)"
{ S7_Optimized_Access := 'TRUE' }
VERSION : 0.1
   VAR_INPUT
      Initial_Call : Bool;   // Initial call of this OB
      Remanence : Bool;   // =True, if remanent data are available
   END_VAR
   VAR_TEMP
      iLastTimeRotation : DTL;
   END_VAR
BEGIN

REGION Network 2
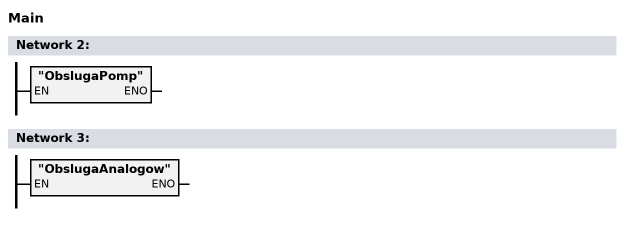
   RUNG wire#powerrail
      "ObslugaPomp"()
   END_RUNG
   // the same network as SCL:
   "ObslugaPomp"();
END_REGION

REGION Network 3
   RUNG wire#powerrail
      "ObslugaAnalogow"()
   END_RUNG
   // the same network as SCL:
   "ObslugaAnalogow"();
END_REGION
END_ORGANIZATION_BLOCK

ORGANIZATION_BLOCK "Startup"   // OB100, LAD, Startup
TITLE = "Complete Restart"
{ S7_Optimized_Access := 'TRUE' }
VERSION : 0.1
   VAR_INPUT
      LostRetentive : Bool;   // True if retentive data are lost
      LostRTC : Bool;   // True if date and time are lost
   END_VAR
   VAR_TEMP
      ret : Int;
   END_VAR
BEGIN

REGION Network 1: Inicjowanie transmisji
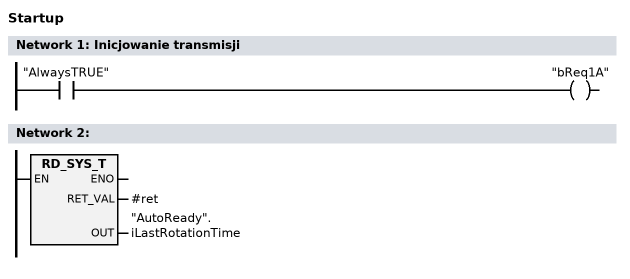
   RUNG wire#powerrail
      Contact( "AlwaysTRUE" )
      Coil( "bReq1A" )
   END_RUNG
   // the same network as SCL:
   "bReq1A" := "AlwaysTRUE";
END_REGION

REGION Network 2
   #ret := RD_SYS_T(OUT => "AutoReady".iLastRotationTime);
END_REGION
END_ORGANIZATION_BLOCK

ORGANIZATION_BLOCK "KomuCycle"   // OB123, LAD, ProgramCycle
TITLE = "Main Program Sweep (Cycle)"
{ S7_Optimized_Access := 'TRUE' }
VERSION : 0.1
   VAR_INPUT
      Initial_Call : Bool;   // Initial call of this OB
      Remanence : Bool;   // =True, if remanent data are available
   END_VAR
   VAR_TEMP
      RS : Bool;
      aTempArr : Array[0..8] of Word;
   END_VAR
   VAR_TEMP   // added for the SCL form of the ladder/FBD networks
      _w1 : Bool;
   END_VAR
BEGIN

REGION Network 1: Zbiornik Kosiby
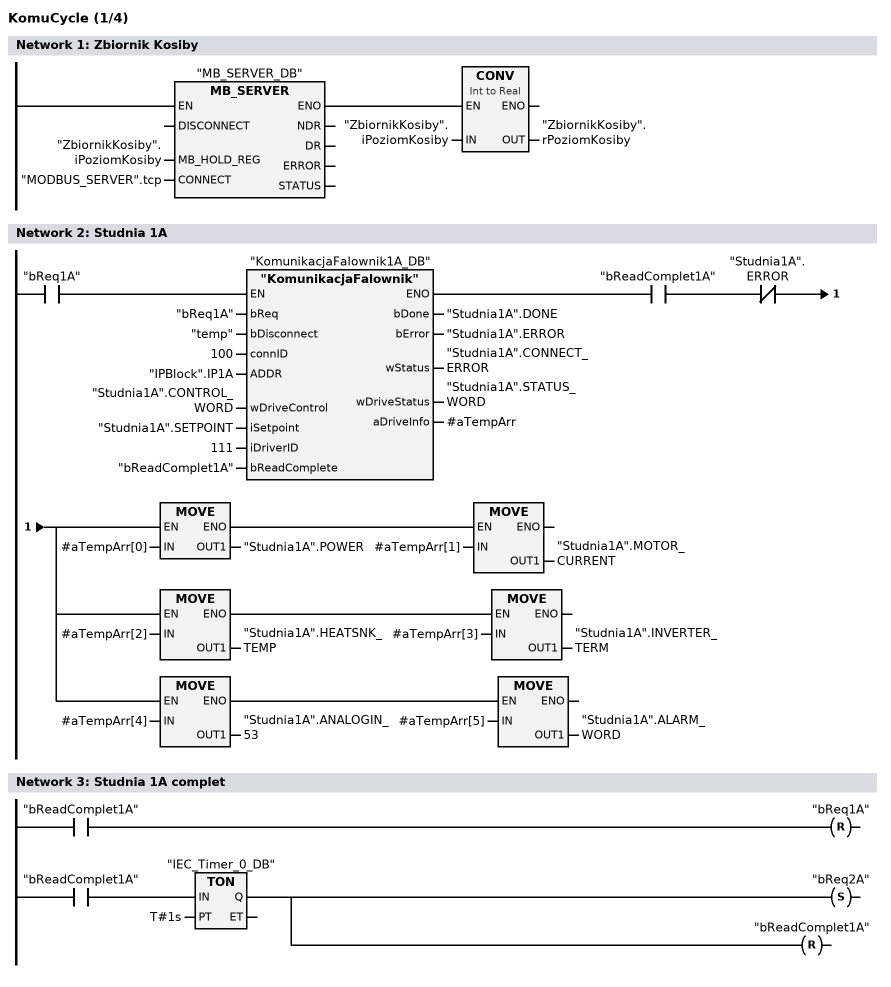
   // ENO of a box is taken as its EN; it also drops when the box reports an error
   "MB_SERVER_DB"(MB_HOLD_REG := "ZbiornikKosiby".iPoziomKosiby, CONNECT := "MODBUS_SERVER".tcp);   // MB_SERVER
   "ZbiornikKosiby".rPoziomKosiby := INT_TO_REAL("ZbiornikKosiby".iPoziomKosiby);
END_REGION

REGION Network 2: Studnia 1A
   RUNG wire#powerrail
      Contact( "bReq1A" )
      "KomunikacjaFalownik1A_DB"(bReq := "bReq1A", bDisconnect := "temp", connID := 100, ADDR := "IPBlock".IP1A, wDriveControl := "Studnia1A".CONTROL_WORD, iSetpoint := "Studnia1A".SETPOINT, iDriverID := 111, bReadComplete := "bReadComplet1A", bDone => "Studnia1A".DONE, bError => "Studnia1A".ERROR, wStatus => "Studnia1A".CONNECT_ERROR, wDriveStatus => "Studnia1A".STATUS_WORD, aDriveInfo => #aTempArr)
      Contact( "bReadComplet1A" )
      I_Contact( "Studnia1A".ERROR )
      wire#w1
      Move(in := #aTempArr[0], out1 => "Studnia1A".POWER)
      Move(in := #aTempArr[1], out1 => "Studnia1A".MOTOR_CURRENT)
   END_RUNG
   RUNG wire#w1
      Move(in := #aTempArr[2], out1 => "Studnia1A".HEATSNK_TEMP)
      Move(in := #aTempArr[3], out1 => "Studnia1A".INVERTER_TERM)
   END_RUNG
   RUNG wire#w1
      Move(in := #aTempArr[4], out1 => "Studnia1A".ANALOGIN_53)
      Move(in := #aTempArr[5], out1 => "Studnia1A".ALARM_WORD)
   END_RUNG
   // the same network as SCL:
   "KomunikacjaFalownik1A_DB"(EN := "bReq1A",   // "KomunikacjaFalownik"
                           bReq := "bReq1A",
                           bDisconnect := "temp",
                           connID := 100,
                           ADDR := "IPBlock".IP1A,
                           wDriveControl := "Studnia1A".CONTROL_WORD,
                           iSetpoint := "Studnia1A".SETPOINT,
                           iDriverID := 111,
                           bReadComplete := "bReadComplet1A",
                           bDone => "Studnia1A".DONE,
                           bError => "Studnia1A".ERROR,
                           wStatus => "Studnia1A".CONNECT_ERROR,
                           wDriveStatus => "Studnia1A".STATUS_WORD,
                           aDriveInfo => #aTempArr,
                           ENO => #_w1);
   IF #_w1 AND "bReadComplet1A" AND NOT "Studnia1A".ERROR THEN
       "Studnia1A".POWER := #aTempArr[0];
       "Studnia1A".MOTOR_CURRENT := #aTempArr[1];
       "Studnia1A".HEATSNK_TEMP := #aTempArr[2];
       "Studnia1A".INVERTER_TERM := #aTempArr[3];
       "Studnia1A".ANALOGIN_53 := #aTempArr[4];
       "Studnia1A".ALARM_WORD := #aTempArr[5];
   END_IF;
END_REGION

REGION Network 3: Studnia 1A complet
   IF "bReadComplet1A" THEN "bReq1A" := FALSE; END_IF;
   "IEC_Timer_0_DB".TON(IN := "bReadComplet1A", PT := T#1s);
   IF "IEC_Timer_0_DB".Q THEN
       "bReq2A" := TRUE;
       "bReadComplet1A" := FALSE;
   END_IF;
END_REGION

REGION Network 4: Studnia 2A kom
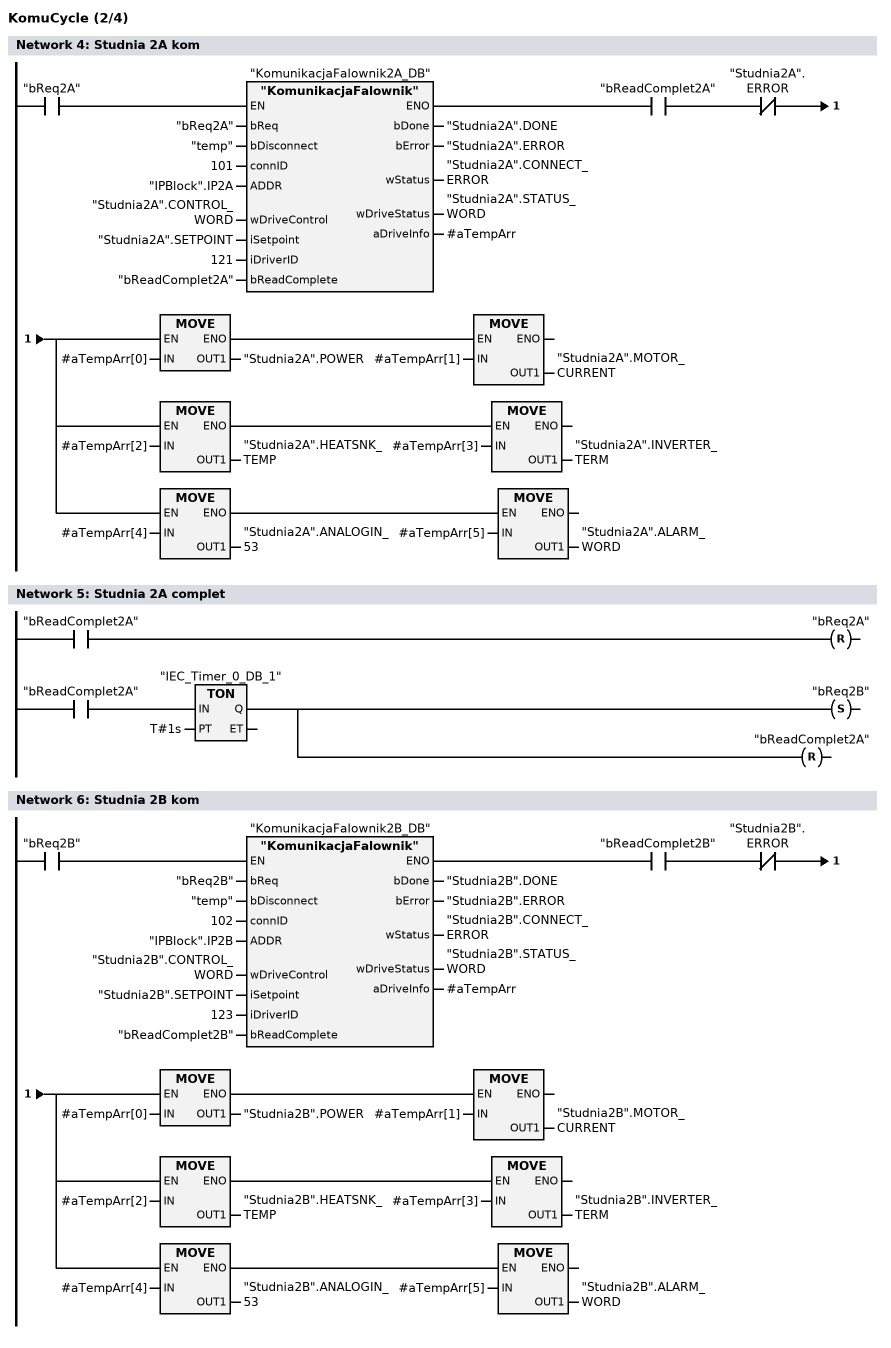
   RUNG wire#powerrail
      Contact( "bReq2A" )
      "KomunikacjaFalownik2A_DB"(bReq := "bReq2A", bDisconnect := "temp", connID := 101, ADDR := "IPBlock".IP2A, wDriveControl := "Studnia2A".CONTROL_WORD, iSetpoint := "Studnia2A".SETPOINT, iDriverID := 121, bReadComplete := "bReadComplet2A", bDone => "Studnia2A".DONE, bError => "Studnia2A".ERROR, wStatus => "Studnia2A".CONNECT_ERROR, wDriveStatus => "Studnia2A".STATUS_WORD, aDriveInfo => #aTempArr)
      Contact( "bReadComplet2A" )
      I_Contact( "Studnia2A".ERROR )
      wire#w1
      Move(in := #aTempArr[0], out1 => "Studnia2A".POWER)
      Move(in := #aTempArr[1], out1 => "Studnia2A".MOTOR_CURRENT)
   END_RUNG
   RUNG wire#w1
      Move(in := #aTempArr[2], out1 => "Studnia2A".HEATSNK_TEMP)
      Move(in := #aTempArr[3], out1 => "Studnia2A".INVERTER_TERM)
   END_RUNG
   RUNG wire#w1
      Move(in := #aTempArr[4], out1 => "Studnia2A".ANALOGIN_53)
      Move(in := #aTempArr[5], out1 => "Studnia2A".ALARM_WORD)
   END_RUNG
   // the same network as SCL:
   "KomunikacjaFalownik2A_DB"(EN := "bReq2A",   // "KomunikacjaFalownik"
                           bReq := "bReq2A",
                           bDisconnect := "temp",
                           connID := 101,
                           ADDR := "IPBlock".IP2A,
                           wDriveControl := "Studnia2A".CONTROL_WORD,
                           iSetpoint := "Studnia2A".SETPOINT,
                           iDriverID := 121,
                           bReadComplete := "bReadComplet2A",
                           bDone => "Studnia2A".DONE,
                           bError => "Studnia2A".ERROR,
                           wStatus => "Studnia2A".CONNECT_ERROR,
                           wDriveStatus => "Studnia2A".STATUS_WORD,
                           aDriveInfo => #aTempArr,
                           ENO => #_w1);
   IF #_w1 AND "bReadComplet2A" AND NOT "Studnia2A".ERROR THEN
       "Studnia2A".POWER := #aTempArr[0];
       "Studnia2A".MOTOR_CURRENT := #aTempArr[1];
       "Studnia2A".HEATSNK_TEMP := #aTempArr[2];
       "Studnia2A".INVERTER_TERM := #aTempArr[3];
       "Studnia2A".ANALOGIN_53 := #aTempArr[4];
       "Studnia2A".ALARM_WORD := #aTempArr[5];
   END_IF;
END_REGION

REGION Network 5: Studnia 2A complet
   IF "bReadComplet2A" THEN "bReq2A" := FALSE; END_IF;
   "IEC_Timer_0_DB_1".TON(IN := "bReadComplet2A", PT := T#1s);
   IF "IEC_Timer_0_DB_1".Q THEN
       "bReq2B" := TRUE;
       "bReadComplet2A" := FALSE;
   END_IF;
END_REGION

REGION Network 6: Studnia 2B kom
   RUNG wire#powerrail
      Contact( "bReq2B" )
      "KomunikacjaFalownik2B_DB"(bReq := "bReq2B", bDisconnect := "temp", connID := 102, ADDR := "IPBlock".IP2B, wDriveControl := "Studnia2B".CONTROL_WORD, iSetpoint := "Studnia2B".SETPOINT, iDriverID := 123, bReadComplete := "bReadComplet2B", bDone => "Studnia2B".DONE, bError => "Studnia2B".ERROR, wStatus => "Studnia2B".CONNECT_ERROR, wDriveStatus => "Studnia2B".STATUS_WORD, aDriveInfo => #aTempArr)
      Contact( "bReadComplet2B" )
      I_Contact( "Studnia2B".ERROR )
      wire#w1
      Move(in := #aTempArr[0], out1 => "Studnia2B".POWER)
      Move(in := #aTempArr[1], out1 => "Studnia2B".MOTOR_CURRENT)
   END_RUNG
   RUNG wire#w1
      Move(in := #aTempArr[2], out1 => "Studnia2B".HEATSNK_TEMP)
      Move(in := #aTempArr[3], out1 => "Studnia2B".INVERTER_TERM)
   END_RUNG
   RUNG wire#w1
      Move(in := #aTempArr[4], out1 => "Studnia2B".ANALOGIN_53)
      Move(in := #aTempArr[5], out1 => "Studnia2B".ALARM_WORD)
   END_RUNG
   // the same network as SCL:
   "KomunikacjaFalownik2B_DB"(EN := "bReq2B",   // "KomunikacjaFalownik"
                           bReq := "bReq2B",
                           bDisconnect := "temp",
                           connID := 102,
                           ADDR := "IPBlock".IP2B,
                           wDriveControl := "Studnia2B".CONTROL_WORD,
                           iSetpoint := "Studnia2B".SETPOINT,
                           iDriverID := 123,
                           bReadComplete := "bReadComplet2B",
                           bDone => "Studnia2B".DONE,
                           bError => "Studnia2B".ERROR,
                           wStatus => "Studnia2B".CONNECT_ERROR,
                           wDriveStatus => "Studnia2B".STATUS_WORD,
                           aDriveInfo => #aTempArr,
                           ENO => #_w1);
   IF #_w1 AND "bReadComplet2B" AND NOT "Studnia2B".ERROR THEN
       "Studnia2B".POWER := #aTempArr[0];
       "Studnia2B".MOTOR_CURRENT := #aTempArr[1];
       "Studnia2B".HEATSNK_TEMP := #aTempArr[2];
       "Studnia2B".INVERTER_TERM := #aTempArr[3];
       "Studnia2B".ANALOGIN_53 := #aTempArr[4];
       "Studnia2B".ALARM_WORD := #aTempArr[5];
   END_IF;
END_REGION

REGION Network 7: Studnia 2B complet
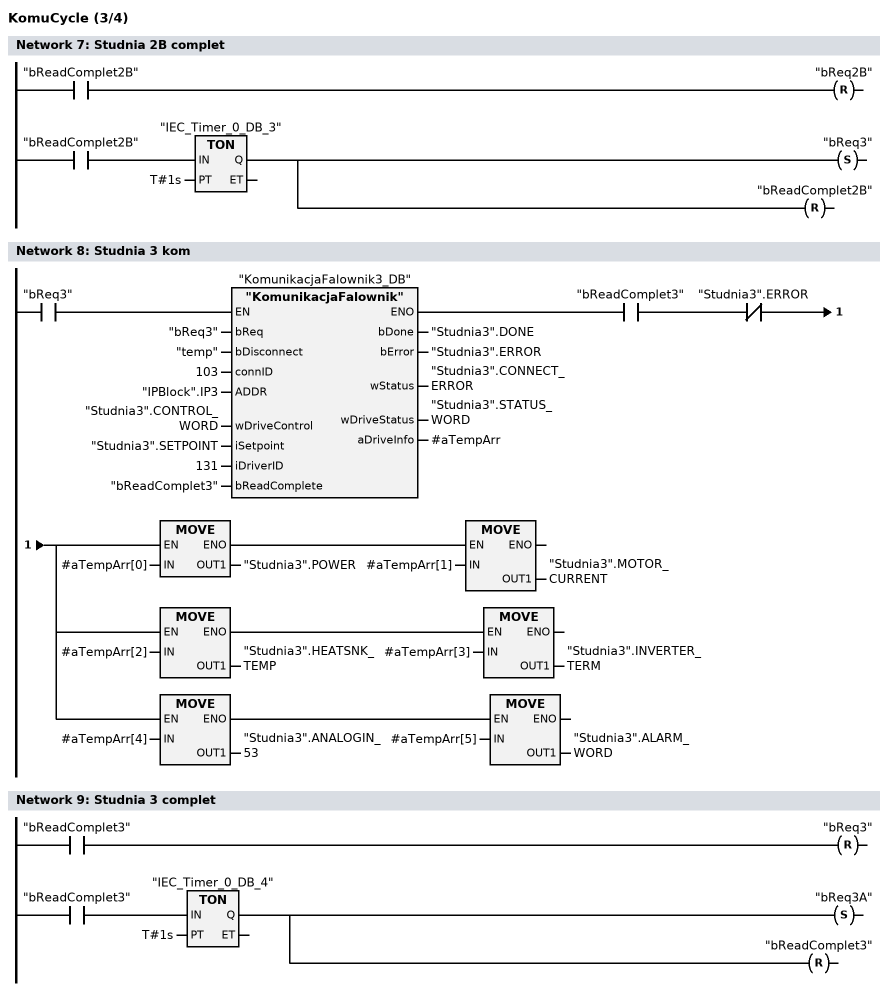
   IF "bReadComplet2B" THEN "bReq2B" := FALSE; END_IF;
   "IEC_Timer_0_DB_3".TON(IN := "bReadComplet2B", PT := T#1s);
   IF "IEC_Timer_0_DB_3".Q THEN
       "bReq3" := TRUE;
       "bReadComplet2B" := FALSE;
   END_IF;
END_REGION

REGION Network 8: Studnia 3 kom
   RUNG wire#powerrail
      Contact( "bReq3" )
      "KomunikacjaFalownik3_DB"(bReq := "bReq3", bDisconnect := "temp", connID := 103, ADDR := "IPBlock".IP3, wDriveControl := "Studnia3".CONTROL_WORD, iSetpoint := "Studnia3".SETPOINT, iDriverID := 131, bReadComplete := "bReadComplet3", bDone => "Studnia3".DONE, bError => "Studnia3".ERROR, wStatus => "Studnia3".CONNECT_ERROR, wDriveStatus => "Studnia3".STATUS_WORD, aDriveInfo => #aTempArr)
      Contact( "bReadComplet3" )
      I_Contact( "Studnia3".ERROR )
      wire#w1
      Move(in := #aTempArr[0], out1 => "Studnia3".POWER)
      Move(in := #aTempArr[1], out1 => "Studnia3".MOTOR_CURRENT)
   END_RUNG
   RUNG wire#w1
      Move(in := #aTempArr[2], out1 => "Studnia3".HEATSNK_TEMP)
      Move(in := #aTempArr[3], out1 => "Studnia3".INVERTER_TERM)
   END_RUNG
   RUNG wire#w1
      Move(in := #aTempArr[4], out1 => "Studnia3".ANALOGIN_53)
      Move(in := #aTempArr[5], out1 => "Studnia3".ALARM_WORD)
   END_RUNG
   // the same network as SCL:
   "KomunikacjaFalownik3_DB"(EN := "bReq3",   // "KomunikacjaFalownik"
                           bReq := "bReq3",
                           bDisconnect := "temp",
                           connID := 103,
                           ADDR := "IPBlock".IP3,
                           wDriveControl := "Studnia3".CONTROL_WORD,
                           iSetpoint := "Studnia3".SETPOINT,
                           iDriverID := 131,
                           bReadComplete := "bReadComplet3",
                           bDone => "Studnia3".DONE,
                           bError => "Studnia3".ERROR,
                           wStatus => "Studnia3".CONNECT_ERROR,
                           wDriveStatus => "Studnia3".STATUS_WORD,
                           aDriveInfo => #aTempArr,
                           ENO => #_w1);
   IF #_w1 AND "bReadComplet3" AND NOT "Studnia3".ERROR THEN
       "Studnia3".POWER := #aTempArr[0];
       "Studnia3".MOTOR_CURRENT := #aTempArr[1];
       "Studnia3".HEATSNK_TEMP := #aTempArr[2];
       "Studnia3".INVERTER_TERM := #aTempArr[3];
       "Studnia3".ANALOGIN_53 := #aTempArr[4];
       "Studnia3".ALARM_WORD := #aTempArr[5];
   END_IF;
END_REGION

REGION Network 9: Studnia 3 complet
   IF "bReadComplet3" THEN "bReq3" := FALSE; END_IF;
   "IEC_Timer_0_DB_4".TON(IN := "bReadComplet3", PT := T#1s);
   IF "IEC_Timer_0_DB_4".Q THEN
       "bReq3A" := TRUE;
       "bReadComplet3" := FALSE;
   END_IF;
END_REGION

REGION Network 10: Studnia 3A kom
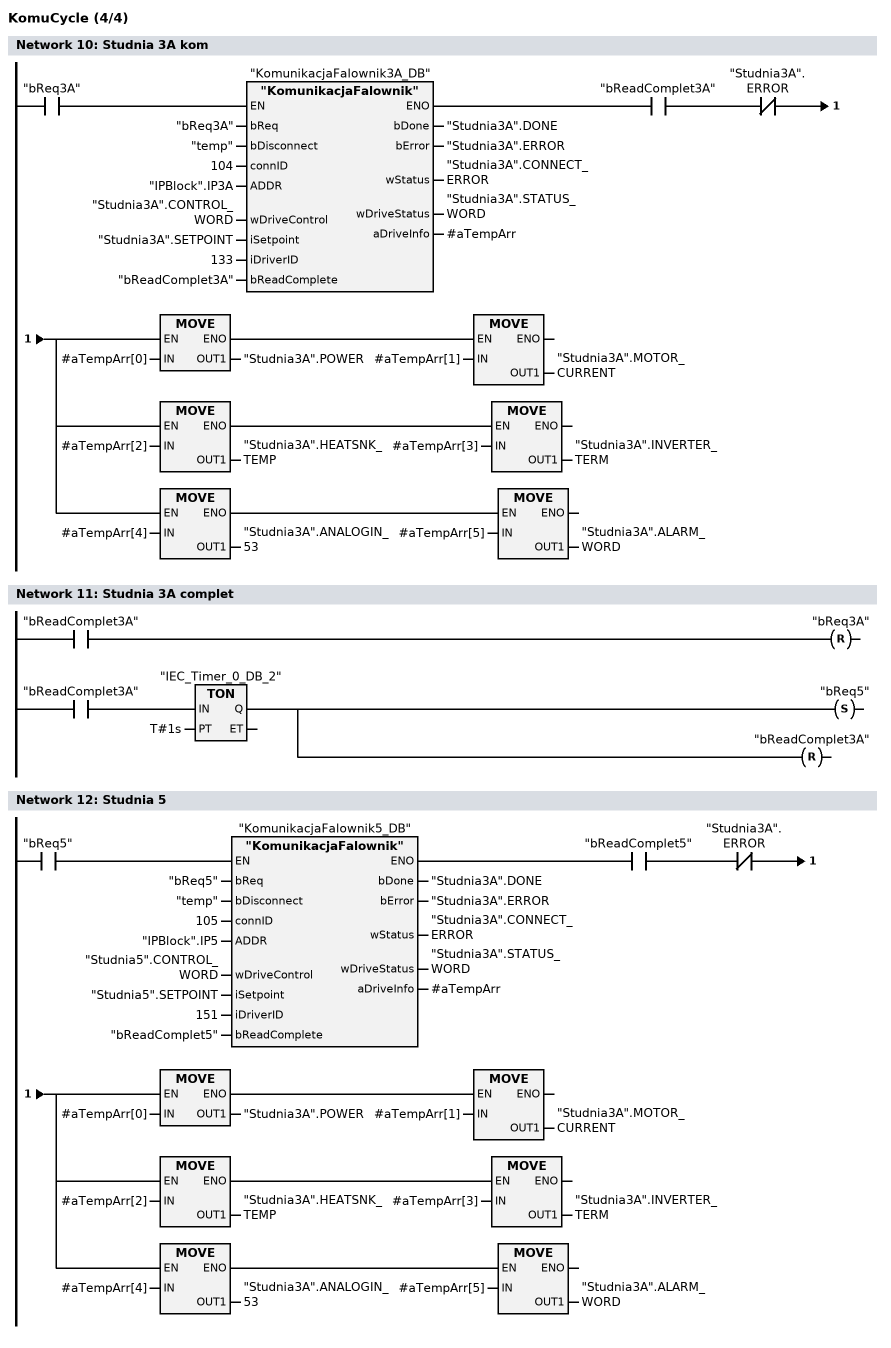
   RUNG wire#powerrail
      Contact( "bReq3A" )
      "KomunikacjaFalownik3A_DB"(bReq := "bReq3A", bDisconnect := "temp", connID := 104, ADDR := "IPBlock".IP3A, wDriveControl := "Studnia3A".CONTROL_WORD, iSetpoint := "Studnia3A".SETPOINT, iDriverID := 133, bReadComplete := "bReadComplet3A", bDone => "Studnia3A".DONE, bError => "Studnia3A".ERROR, wStatus => "Studnia3A".CONNECT_ERROR, wDriveStatus => "Studnia3A".STATUS_WORD, aDriveInfo => #aTempArr)
      Contact( "bReadComplet3A" )
      I_Contact( "Studnia3A".ERROR )
      wire#w1
      Move(in := #aTempArr[0], out1 => "Studnia3A".POWER)
      Move(in := #aTempArr[1], out1 => "Studnia3A".MOTOR_CURRENT)
   END_RUNG
   RUNG wire#w1
      Move(in := #aTempArr[2], out1 => "Studnia3A".HEATSNK_TEMP)
      Move(in := #aTempArr[3], out1 => "Studnia3A".INVERTER_TERM)
   END_RUNG
   RUNG wire#w1
      Move(in := #aTempArr[4], out1 => "Studnia3A".ANALOGIN_53)
      Move(in := #aTempArr[5], out1 => "Studnia3A".ALARM_WORD)
   END_RUNG
   // the same network as SCL:
   "KomunikacjaFalownik3A_DB"(EN := "bReq3A",   // "KomunikacjaFalownik"
                           bReq := "bReq3A",
                           bDisconnect := "temp",
                           connID := 104,
                           ADDR := "IPBlock".IP3A,
                           wDriveControl := "Studnia3A".CONTROL_WORD,
                           iSetpoint := "Studnia3A".SETPOINT,
                           iDriverID := 133,
                           bReadComplete := "bReadComplet3A",
                           bDone => "Studnia3A".DONE,
                           bError => "Studnia3A".ERROR,
                           wStatus => "Studnia3A".CONNECT_ERROR,
                           wDriveStatus => "Studnia3A".STATUS_WORD,
                           aDriveInfo => #aTempArr,
                           ENO => #_w1);
   IF #_w1 AND "bReadComplet3A" AND NOT "Studnia3A".ERROR THEN
       "Studnia3A".POWER := #aTempArr[0];
       "Studnia3A".MOTOR_CURRENT := #aTempArr[1];
       "Studnia3A".HEATSNK_TEMP := #aTempArr[2];
       "Studnia3A".INVERTER_TERM := #aTempArr[3];
       "Studnia3A".ANALOGIN_53 := #aTempArr[4];
       "Studnia3A".ALARM_WORD := #aTempArr[5];
   END_IF;
END_REGION

REGION Network 11: Studnia 3A complet
   IF "bReadComplet3A" THEN "bReq3A" := FALSE; END_IF;
   "IEC_Timer_0_DB_2".TON(IN := "bReadComplet3A", PT := T#1s);
   IF "IEC_Timer_0_DB_2".Q THEN
       "bReq5" := TRUE;
       "bReadComplet3A" := FALSE;
   END_IF;
END_REGION

REGION Network 12: Studnia 5
   RUNG wire#powerrail
      Contact( "bReq5" )
      "KomunikacjaFalownik5_DB"(bReq := "bReq5", bDisconnect := "temp", connID := 105, ADDR := "IPBlock".IP5, wDriveControl := "Studnia5".CONTROL_WORD, iSetpoint := "Studnia5".SETPOINT, iDriverID := 151, bReadComplete := "bReadComplet5", bDone => "Studnia3A".DONE, bError => "Studnia3A".ERROR, wStatus => "Studnia3A".CONNECT_ERROR, wDriveStatus => "Studnia3A".STATUS_WORD, aDriveInfo => #aTempArr)
      Contact( "bReadComplet5" )
      I_Contact( "Studnia3A".ERROR )
      wire#w1
      Move(in := #aTempArr[0], out1 => "Studnia3A".POWER)
      Move(in := #aTempArr[1], out1 => "Studnia3A".MOTOR_CURRENT)
   END_RUNG
   RUNG wire#w1
      Move(in := #aTempArr[2], out1 => "Studnia3A".HEATSNK_TEMP)
      Move(in := #aTempArr[3], out1 => "Studnia3A".INVERTER_TERM)
   END_RUNG
   RUNG wire#w1
      Move(in := #aTempArr[4], out1 => "Studnia3A".ANALOGIN_53)
      Move(in := #aTempArr[5], out1 => "Studnia3A".ALARM_WORD)
   END_RUNG
   // the same network as SCL:
   "KomunikacjaFalownik5_DB"(EN := "bReq5",   // "KomunikacjaFalownik"
                           bReq := "bReq5",
                           bDisconnect := "temp",
                           connID := 105,
                           ADDR := "IPBlock".IP5,
                           wDriveControl := "Studnia5".CONTROL_WORD,
                           iSetpoint := "Studnia5".SETPOINT,
                           iDriverID := 151,
                           bReadComplete := "bReadComplet5",
                           bDone => "Studnia3A".DONE,
                           bError => "Studnia3A".ERROR,
                           wStatus => "Studnia3A".CONNECT_ERROR,
                           wDriveStatus => "Studnia3A".STATUS_WORD,
                           aDriveInfo => #aTempArr,
                           ENO => #_w1);
   IF #_w1 AND "bReadComplet5" AND NOT "Studnia3A".ERROR THEN
       "Studnia3A".POWER := #aTempArr[0];
       "Studnia3A".MOTOR_CURRENT := #aTempArr[1];
       "Studnia3A".HEATSNK_TEMP := #aTempArr[2];
       "Studnia3A".INVERTER_TERM := #aTempArr[3];
       "Studnia3A".ANALOGIN_53 := #aTempArr[4];
       "Studnia3A".ALARM_WORD := #aTempArr[5];
   END_IF;
END_REGION
END_ORGANIZATION_BLOCK